(* Logix 5000 project; controller DUNEW2PLC1 vendor 1 type 14 code 221 rev 33.11; software revision 33.00 *)

TASK DUNEWINDER2 (continuous, watchdog 500 ms) : MainProgram, UnServo_9, EOT_Trip_11, Error_State_10, Latch_UnLatch_State_6_7_8, MoveXY_State_2_3, MoveZ_State_4_5, Ready_State_1, Initialize, PID_Tension_Servo
TASK SafetyTask (periodic, rate 20 ms, priority 10, watchdog 20 ms) : Safety

MODULES
   Local : vendor 1 type 14 code 221 (5069 0, rev 33.11)
      DUNEW2AMP : 2198-P031 (Ethernet 192.168.140.15, rev 11.3, A_MotionDiagnostics RPI 1 ms, B_MotionSync RPI 2 ms)
      DUNEW2SERVO2 : vendor 1 type 45 code 31 (Ethernet 192.168.140.17, rev 11.2, C_Safety_Output RPI 20 ms, B_MotionSync RPI 2 ms, D_Safety_Input RPI 10 ms, A_MotionDiagnostics RPI 1 ms)
      DUNEW2SERVO1 : vendor 1 type 45 code 31 (Ethernet 192.168.140.16, rev 11.3, C_Safety_Output RPI 20 ms, A_MotionDiagnostics RPI 1 ms, D_Safety_Input RPI 10 ms, B_MotionSync RPI 2 ms)
      DUNEW2NETSW : vendor 1 type 12 code 241 (Ethernet 192.168.140.10, rev 10.1, Output RPI 1000 ms)
      DUNE2CAM1 : vendor 678 type 100 code 274 (Ethernet 192.168.140.19, rev 11.1, Output RPI 60 ms)
       : vendor 1 type 115 code 313 (5069 5, rev 2.1, StandardDataDriven RPI 13.1 ms)
           Local:5:O.Ch00.Data   // Tension_Servo_CMD
       : 5069-IB16 (5069 2, rev 2.14, StandardDataDriven RPI 5 ms)
           Local:2:I.Pt07.Data   // O/T SWITCH OVERTRAVEL SWITCH
           Local:2:I.Pt06.Data   // TENSION ON/OFF
           Local:2:I.Pt13.Data   // Cabinet lighted push button
       : 5069-IB16 (5069 6, rev 2.14, StandardDataDriven RPI 5 ms)
       : 5069-OB16 (5069 3, rev 2.14, StandardDataDriven RPI 5 ms)
           Local:3:O.Pt01.Data   // Latching signal output
           Local:3:O.Pt11.Data   // Reset PB - Light
           Local:3:O.Pt15.Data   // Beacon - Sounder
           Local:3:O.Pt13.Data   // Beacon - Amber
           Local:3:O.Pt12.Data   // Beacon - Green
           Local:3:O.Pt14.Data   // Beacon - Red
       : 5069-OB16 (5069 7, rev 2.14, StandardDataDriven RPI 5 ms)
       : 5069-IF8 (5069 4, rev 2.11, StandardDataDriven RPI 12.5 ms)
           Local:4:I   // Wire tension (N)
       : 5069-IB16 (5069 1, rev 2.14, StandardDataDriven RPI 5 ms)
           Local:1:I.Pt08.Data   // Latch top
           Local:1:I.Pt15.Data   // The wire break switch was causing electrical problems, so we use the load-cell as a proxy for wire break
           Local:1:I.Pt09.Data   // Latch middle
      DUNEW2PLC2 : 1734-AENT (Ethernet 192.168.140.14, rev 6.12)
          : vendor 1 type 35 code 16 (PointIO 2, rev 2.1, Output RPI 20 ms, Input RPI 10 ms)
          : vendor 1 type 35 code 15 (PointIO 1, rev 2.1, Output RPI 20 ms, Input RPI 10 ms)
              DUNEW2PLC2:1:I.Pt03Data   // EStop Pullcord 1
              DUNEW2PLC2:1:I.Pt04Data   // EStop Pullcord 2
              DUNEW2PLC2:1:I.Pt02Data   // EStop Rack
              DUNEW2PLC2:1:I.Pt01Data   // LC OSS2
              DUNEW2PLC2:1:I.Pt05Data   // Run Key
              DUNEW2PLC2:1:I.Pt00Data   // LC OSS1
END_MODULES

ADD_ON_INSTRUCTION SCP   (* revision 1.0, vendor CVKI *)
// Scale with Parameters
// Help:
// Rockwell Software RSLogix 500 Description:
// The Input value is scaled to a range determined by creating a linear relationship between input min and max values and scaled min and max values. The scaled result is returned to the address indicated by the output parameter.
VAR_INPUT
   Input : REAL; {required}   // Value to be Scaled
   Input_Min : REAL; {required}   // Minimum Value for the Input
   Input_Max : REAL; {required}   // Maximum Value for the Input
   Scaled_Min : REAL; {required}   // Minimum Scaling Value
   Scaled_Max : REAL; {required}   // Maximum Scaling Value
END_VAR
VAR_OUTPUT
   Output : REAL; {access Read Only, required}   // Scaled Value [Slope*Input + Offset]
END_VAR
VAR
   offset : REAL;   // Offset Value [Scaled Min - (Input Min * Slope)]
   slope : REAL;   // Slope Value [(Scaled Max - Scaled Min)/(Input Max - Input Min)]
END_VAR

ROUTINE Logic   (* ladder *)
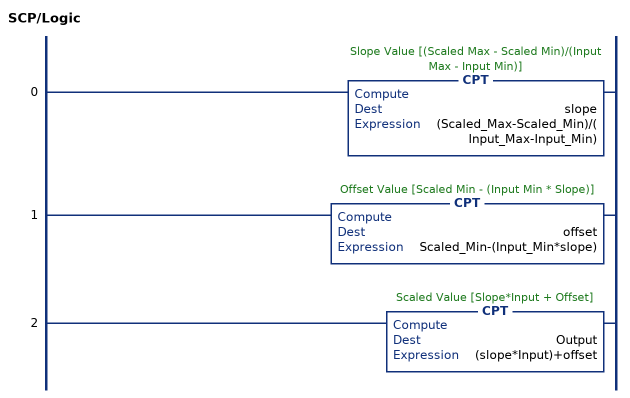
   0: CPT(slope,(Scaled_Max-Scaled_Min)/(Input_Max-Input_Min));
   1: CPT(offset,Scaled_Min-(Input_Min*slope));
   2: CPT(Output,(slope*Input)+offset);
END_ROUTINE
END_ADD_ON_INSTRUCTION

VAR_GLOBAL   (* controller tags *)
   a_actual : REAL := 700.0062;
   a_signed : REAL := -243.85713;
   accel_xy : REAL;   // Tangential acceleration of the winding head in xy-plane
   ACTUATOR_POS : DINT := 1; {access Read Only}
   AFI : BOOL;
   ALL_EOT_GOOD : BOOL := 1; {access Read Only}
   always_regulate_speed : BOOL := 1;
   APA_IS_VERTICAL : BOOL; {access Read Only}
   blink_off : TIMER := (PRE := 500, ACC := 490, EN := 1, TT := 1);
   blink_on : TIMER := (PRE := 500, ACC := 500, EN := 1, DN := 1);
   bypass_xy_move : BOOL := 1;
   CAM_F_EN : BOOL := 1;
   CAM_F_TRIGGER : BOOL := 1;
   check_tension_stable : BOOL := 1;   // Check if the tension is stable at the setpoint before moving the winding head
   current_command : REAL;
   current_command_high : REAL := 1.5; {constant}
   current_command_low : REAL := -0.5; {constant}
   DUNEW1AMP : AXIS_CIP_DRIVE;
   DUNEW2AXIS : MOTION_GROUP;
   EN_POS_TRIGGERS : BOOL;
   Enable_SFX : BOOL;
   Enable_SLS : BOOL;
   ERROR_CODE : DINT; {access Read Only}
   ESTOP : ALIAS FOR DUNEW2PLC2:1:I.Pt02Data;
   FIFO_Data : REAL[6]; {access Read Only}
   FIFO_FLUSH : BOOL;   // Flush the camera FIFOs.
   FRAME_LOC_FT_BTM : BOOL := 1;
   FRAME_LOC_FT_MID : BOOL := 1;
   FRAME_LOC_FT_TOP : BOOL := 1;
   FRAME_LOC_HD_BTM : BOOL := 1;
   FRAME_LOC_HD_MID : BOOL := 1;
   FRAME_LOC_HD_TOP : BOOL := 1;
   gamma : REAL := 20.0;
   HEAD_POS : DINT;
   HomeTrigger : BOOL;
   INIT_DONE : BOOL := 1; {access Read Only}
   INPUTS2 : ALIAS FOR Local:2:I;
   J : REAL := 2000.0;
   LATCH_ACTUATOR_BOTTOM : BOOL;
   LATCH_ACTUATOR_HOMED : BOOL; {access Read Only}
   LATCH_ACTUATOR_MID : BOOL;
   LATCH_ACTUATOR_TOP : BOOL;
   latch_ouput : ALIAS FOR Local:3:O.Pt01.Data;
   MACHINE_SW_STAT : BOOL[32] := ([1] := 1, [2] := 1, [3] := 1, [4] := 1, [6] := 1, [8] := 1, [9] := 1, [17] := 1, [18] := 1, [19] := 1, [20] := 1, [21] := 1, [25] := 1, [26] := 1, [27] := 1, [28] := 1, [29] := 1, [30] := 1, [31] := 1); {access Read Only}
   MAS : BOOL := 1;   // Motion Axis Stop
   MASTER_Z_GO : BOOL := 1; {access Read Only}
   max_tolerable_tension : REAL := 9.0;
   MAX_TOLERABLE_Z : REAL := 5.0; {constant}
   MCCD_X_Y_Axis : MOTION_INSTRUCTION := (FLAGS := 33554432);
   MCCD_X_Y_Axis1 : MOTION_INSTRUCTION := (FLAGS := 33554432);
   MINUS_X_EOT : BOOL := 1; {access Read Only}
   MINUS_Y_EOT : BOOL := 1; {access Read Only}
   MORE_STATS : BOOL[32]; {access Read Only}
   MORE_STATS_S : BOOL[32] := ([0] := 1);
   MOVE_TYPE : INT;   // 0 = No Move 1 = XY JOG 2 = XY Plane Move 3 = Z JOG 4 = Z Axis Move 5 = Toggle Latch Actuator 6 = Home the Latch Actuator 7 = Unlock Latch Actuator Motor 8 = Un-Servo Motors 9 = PLC_Init
   neutral_cv : REAL := 2.5;
   NEXTSTATE : DINT := 1; {access Read Only}
   overtension_timer : TIMER := (PRE := 100);
   pid_cv_high_limit : REAL := 10.0;
   pid_cv_low_limit : REAL;
   pid_cv_out : REAL := 2.5;
   PID_LOOP_TIMER : TIMER := (PRE := 5, ACC := 4, EN := 1, TT := 1);
   pid_loop_timer_bypass : BOOL;
   pid_start_bias : BOOL;
   PLUS_X_EOT : BOOL := 1; {access Read Only}
   PLUS_Y_EOT : BOOL := 1; {access Read Only}
   POSITION : REAL[1,2]; {constant}
   READ_FIFOS : BOOL;
   ResetPB : BOOL;
   resetPB_S : BOOL;
   ROT_LOC_KEY : AB:1769_DI32:I:0; {access Read Only}
   Run_Alarm : BOOL;
   Safety_Reset_FallingEdge : BOOL;
   Safety_System_Healthy : BOOL := 1;
   Safety_Tripped_S : BOOL;
   SetPoint_CV : REAL;
   SetPoint_Override : REAL;
   SetPoint_PV : REAL := 2.3567553;   // wire tension from load cell (N)
   SLS_Active_Limit : REAL := 50.0;
   SLS_Request1 : BOOL;
   speed_regulator_switch : BOOL := 1;   // This is our "enable safe speed" switch, repurposed to switch the speed regulator
   STATE : DINT := 1; {access Read Only}   // CURRENT State Machine State
   STATE6_IND : BOOL; {access Read Only}
   STATE8_IND : BOOL := 1; {access Read Only}
   T01 : TIMER := (PRE := 5000, ACC := 5000, EN := 1, DN := 1);
   tension : ALIAS FOR Local:4:I.Ch01.Data;   // wire tension (N)
   TENSION_CONTROL_OK : BOOL;
   tension_limited_speed : REAL;
   tension_motor_out : ALIAS FOR Local:5:O.Ch00.Data;
   TENSION_ON_SWITCH : BOOL;
   tension_on_switch_delay_on_start : TIMER := (PRE := 1000);
   tension_setpoint : REAL := 6.25;
   tension_stabilizing : BOOL := 1;
   tension_stable_timer : TIMER := (PRE := 200);
   v_0 : REAL := 0.049999997;
   v_xy : REAL;   // velocity of winding head in xy plane
   v_xyz : REAL;   // Velocity of winding head in xyz space
   winding_head_pid : PID := (CTL := 41984, INI := 1, OLL := 1, DVNA := 1, SP := 2.0, KP := 0.1, KI := 0.4, KD := 0.1, MAXS := 10.0, MAXO := 100.0, UPD := 0.05, PV := 2.3567543, ERR := -0.3567543, PVH := 10.0, MAXI := 10.0, MAXCV := 10.0, MAXTIE := 10.0, DATA[0] := 0.20484047, DATA[1] := -377.08075, DATA[2] := 2.3567543, DATA[3] := -0.3567543, DATA[4] := 2.0, DATA[5] := 10.0, DATA[6] := 1.0, DATA[7] := 0.90000004, DATA[8] := 0.1, DATA[9] := 0.4, DATA[10] := 0.1, DATA[11] := 0.1, DATA[12] := 0.4, DATA[13] := 0.1, DATA[15] := 0.1, DATA[16] := 10.0);
   wire_break_proxy : BOOL;
   wire_break_tension : REAL := 2.5;
   X_axis : AXIS_CIP_DRIVE; {access Read Only}
   X_Axis_SFX : SAFETY_FEEDBACK_INTERFACE := (FeedbackValid := 1, O1 := 1, PositionScaling := 512.0, FeedbackResolution := 512, Unwind := 512, FaultType := 1, PositionScalingOut := 512.0, UnwindOut := 512);
   X_Axis_SLS : SAFELY_LIMITED_SPEED := (RestartType := 1, ColdStartType := 1, O1 := 1, CheckDelay := 3000, ActiveLimit := 10.0, FaultType := 1);
   X_DELTA : REAL;
   X_PARKED : BOOL; {access Read Only}
   X_POSITION : ALIAS FOR POSITION[0,0]; {constant}
   X_SPEED : REAL;
   X_XFER_OK : BOOL; {access Read Only}   // If at the head, check head support arms. Same for foot
   X_Y : COORDINATE_SYSTEM;
   XY_ACCELERATION : REAL := 150.0;   // Maximum positive acceleration for position move.
   XY_DECEL_REQ : REAL;
   XY_DECELERATION : REAL := 300.0;   // Maximum negative acceleration for position move.
   XY_MAX_ACCELERATION : REAL;   // Maximum positive acceleration for position move.
   XY_MAX_DECELERATION : REAL;   // Maximum negative acceleration for position move.
   XY_MAX_VELOCITY : REAL;   // Maximum velocity for position move.
   xy_regulated_acceleration : REAL := 2000.0;
   xy_regulated_deceleration : REAL := 2000.0;
   XY_SPEED : REAL := 300.0;   // Maximum velocity for position move.
   XY_SPEED_REQ : REAL := 300.0;   // XY Requested speed copy of XY_Speed to be used for MCLM and MCCD in MoveXY
   Y_axis : AXIS_CIP_DRIVE; {access Read Only}
   Y_DELTA : REAL := 5.75;
   Y_MOUNT_XFER_OK : BOOL; {access Read Only}
   Y_POSITION : ALIAS FOR POSITION[0,1]; {constant}
   Y_SPEED : REAL;
   Y_XFER_OK : BOOL := 1; {access Read Only}
   Y_Xfer_Window_Btm : BOOL;
   Y_Xfer_Window_Mid : BOOL;
   Y_Xfer_Window_Top : BOOL;
   Z_ACCELERATION : REAL := 600.0;
   Z_axis : AXIS_CIP_DRIVE; {access Read Only}
   Z_DECELLERATION : REAL := 600.0;
   Z_EOT : BOOL := 1; {access Read Only}
   Z_EXTENDED : BOOL; {access Read Only}
   Z_FIXED_LATCHED : BOOL; {access Read Only}
   Z_FIXED_PRESENT : BOOL; {access Read Only}
   Z_OK_TO_ENGAGE : BOOL; {access Read Only}
   Z_POSITION : REAL;
   Z_RETRACTED : BOOL := 1; {access Read Only}
   Z_SAFE_TO_WITHDRAW : BOOL;
   Z_SPEED : REAL;
   Z_STAGE_LATCHED : BOOL := 1; {access Read Only}
   Z_STAGE_PRESENT : BOOL := 1; {access Read Only}   // Winding head is on the Z-arm
   Z_STAGE_UNLATCHED : BOOL; {access Read Only}
END_VAR

PROGRAM Camera   (* main routine CameraControl *)
// Controls to capture data from the Cognex camera.
VAR
   Cam_F_InspectionRes_0 : REAL[32]; {access Read Only}
   Cam_F_InspectionRes_1 : REAL[10]; {access Read Only}
   Cam_F_InspectionRes_2 : REAL[10]; {access Read Only}
   Cam_F_InspectionRes_3 : REAL[10]; {access Read Only}
   FIFO_CTRL : CONTROL[6] := ([0].LEN := 10, [0].EM := 1, [1].LEN := 10, [1].EM := 1, [2].LEN := 10, [2].EM := 1, [3].LEN := 10, [3].EM := 1, [4].LEN := 10, [4].EM := 1, [5].LEN := 10, [5].EM := 1); {access Read Only}
   foundIt : BOOL; {access Read Only}
   LightRing : TIMER := (PRE := 100); {access Read Only}
   Manual_Trig : BOOL; {access Read Only}
   osob : BOOL[32]; {access Read Only}
   ossb : BOOL[32] := ([3] := 1); {access Read Only}
   Pos_trigger : BOOL := 1; {access Read Only}
   RegistrationData : MOTION_INSTRUCTION[8] := ([0].FLAGS := -1845493760, [0].EN := 1, [0].ER := 1, [0].ERR := 3, [1].FLAGS := -1845493760, [1].EN := 1, [1].ER := 1, [1].ERR := 3); {access Read Only}
   triggerOneShotOB : BOOL; {access Read Only}
   triggerOneShotSB : BOOL := 1; {access Read Only}
   TriggerResetTimer1 : TIMER := (PRE := 100, ACC := 5, EN := 1, TT := 1); {access Read Only}
   TriggerResetTimer2 : TIMER := (PRE := 100); {access Read Only}
   X_axis_Cam_F_Pos : REAL[10]; {access Read Only}
   X_axis_Cam_F_Position : REAL := -5.1799655; {access Read Only}
   x_pos : REAL := 564.005; {access Read Only}
   x_pos_next : REAL := 564.005;
   Y_axis_Cam_F_Pos : REAL[10]; {access Read Only}
   Y_axis_Cam_F_Position : REAL := 12.123628; {access Read Only}
   y_pos : REAL := 2465.8398;
   y_pos_next : REAL := 2465.8398;
END_VAR

ROUTINE CameraControl   (* ladder *)
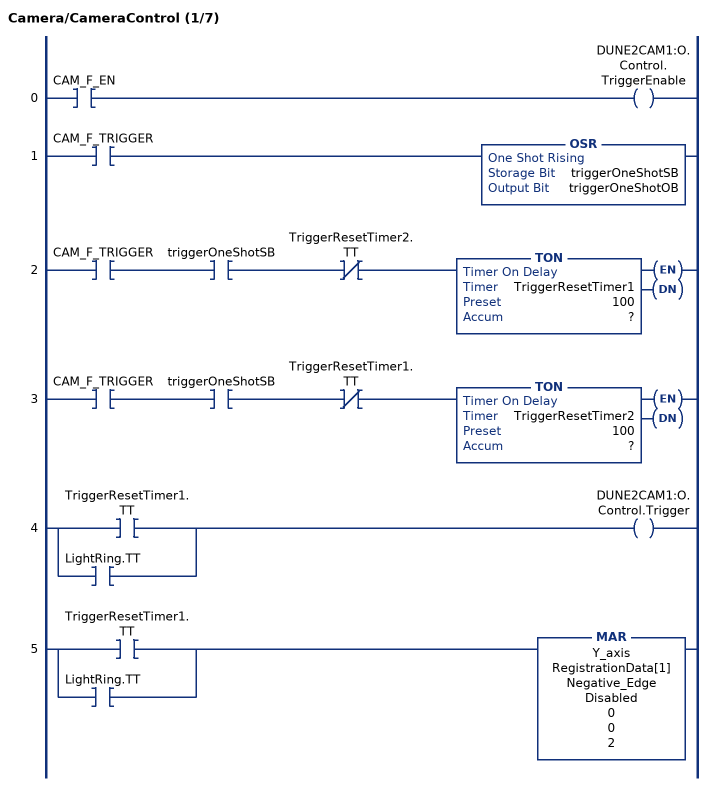
   0: XIC(CAM_F_EN)OTE(DUNE2CAM1:O.Control.TriggerEnable);
   1: XIC(CAM_F_TRIGGER)OSR(triggerOneShotSB,triggerOneShotOB);
   2: XIC(CAM_F_TRIGGER)XIC(triggerOneShotSB)XIO(TriggerResetTimer2.TT)TON(TriggerResetTimer1,?,?);
   3: XIC(CAM_F_TRIGGER)XIC(triggerOneShotSB)XIO(TriggerResetTimer1.TT)TON(TriggerResetTimer2,?,?);
   4: [XIC(TriggerResetTimer1.TT) ,XIC(LightRing.TT) ]OTE(DUNE2CAM1:O.Control.Trigger);
   5: [XIC(TriggerResetTimer1.TT) ,XIC(LightRing.TT) ]MAR(Y_axis,RegistrationData[1],Negative_Edge,Disabled,0,0,2);
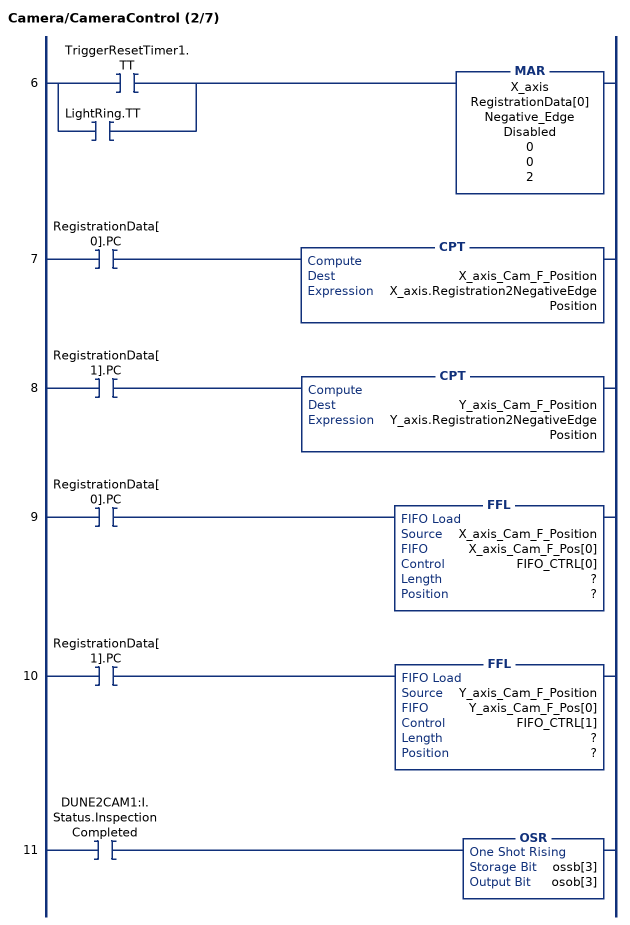
   6: [XIC(TriggerResetTimer1.TT) ,XIC(LightRing.TT) ]MAR(X_axis,RegistrationData[0],Negative_Edge,Disabled,0,0,2);
   7: XIC(RegistrationData[0].PC)CPT(X_axis_Cam_F_Position,X_axis.Registration2NegativeEdgePosition);
   8: XIC(RegistrationData[1].PC)CPT(Y_axis_Cam_F_Position,Y_axis.Registration2NegativeEdgePosition);
   9: XIC(RegistrationData[0].PC)FFL(X_axis_Cam_F_Position,X_axis_Cam_F_Pos[0],FIFO_CTRL[0],?,?);
   10: XIC(RegistrationData[1].PC)FFL(Y_axis_Cam_F_Position,Y_axis_Cam_F_Pos[0],FIFO_CTRL[1],?,?);
   11: XIC(DUNE2CAM1:I.Status.InspectionCompleted)OSR(ossb[3],osob[3]);
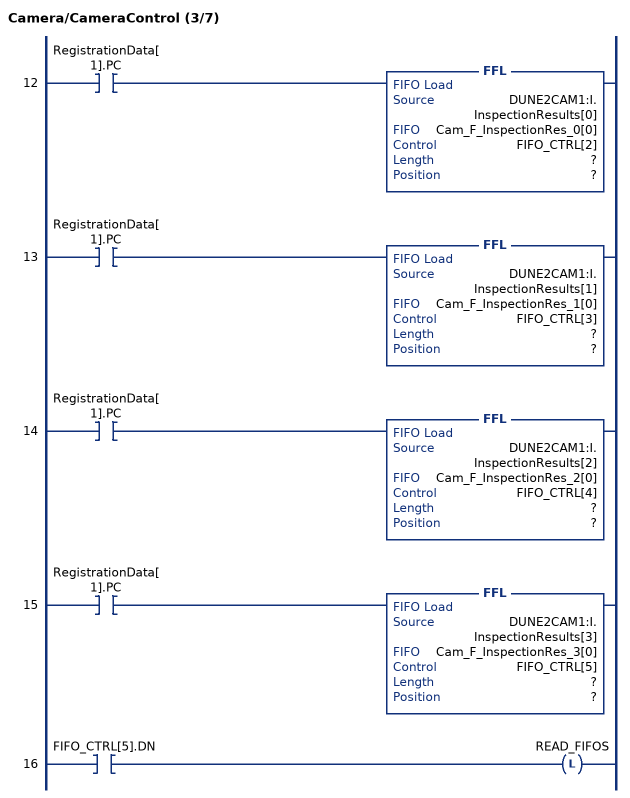
   12: XIC(RegistrationData[1].PC)FFL(DUNE2CAM1:I.InspectionResults[0],Cam_F_InspectionRes_0[0],FIFO_CTRL[2],?,?);
   13: XIC(RegistrationData[1].PC)FFL(DUNE2CAM1:I.InspectionResults[1],Cam_F_InspectionRes_1[0],FIFO_CTRL[3],?,?);
   14: XIC(RegistrationData[1].PC)FFL(DUNE2CAM1:I.InspectionResults[2],Cam_F_InspectionRes_2[0],FIFO_CTRL[4],?,?);
   15: XIC(RegistrationData[1].PC)FFL(DUNE2CAM1:I.InspectionResults[3],Cam_F_InspectionRes_3[0],FIFO_CTRL[5],?,?);
   16: XIC(FIFO_CTRL[5].DN)OTL(READ_FIFOS);
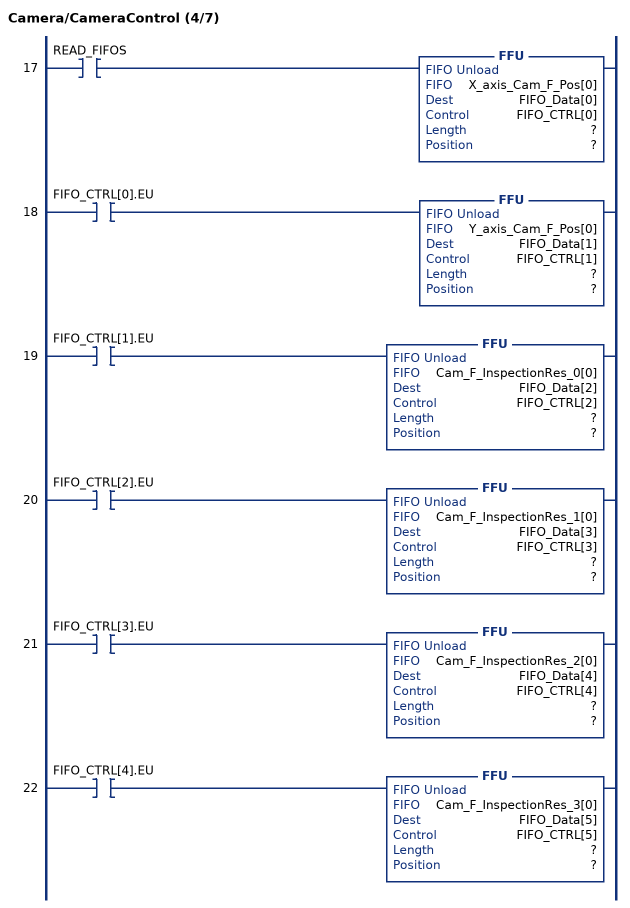
   17: XIC(READ_FIFOS)FFU(X_axis_Cam_F_Pos[0],FIFO_Data[0],FIFO_CTRL[0],?,?);
   18: XIC(FIFO_CTRL[0].EU)FFU(Y_axis_Cam_F_Pos[0],FIFO_Data[1],FIFO_CTRL[1],?,?);
   19: XIC(FIFO_CTRL[1].EU)FFU(Cam_F_InspectionRes_0[0],FIFO_Data[2],FIFO_CTRL[2],?,?);
   20: XIC(FIFO_CTRL[2].EU)FFU(Cam_F_InspectionRes_1[0],FIFO_Data[3],FIFO_CTRL[3],?,?);
   21: XIC(FIFO_CTRL[3].EU)FFU(Cam_F_InspectionRes_2[0],FIFO_Data[4],FIFO_CTRL[4],?,?);
   22: XIC(FIFO_CTRL[4].EU)FFU(Cam_F_InspectionRes_3[0],FIFO_Data[5],FIFO_CTRL[5],?,?);
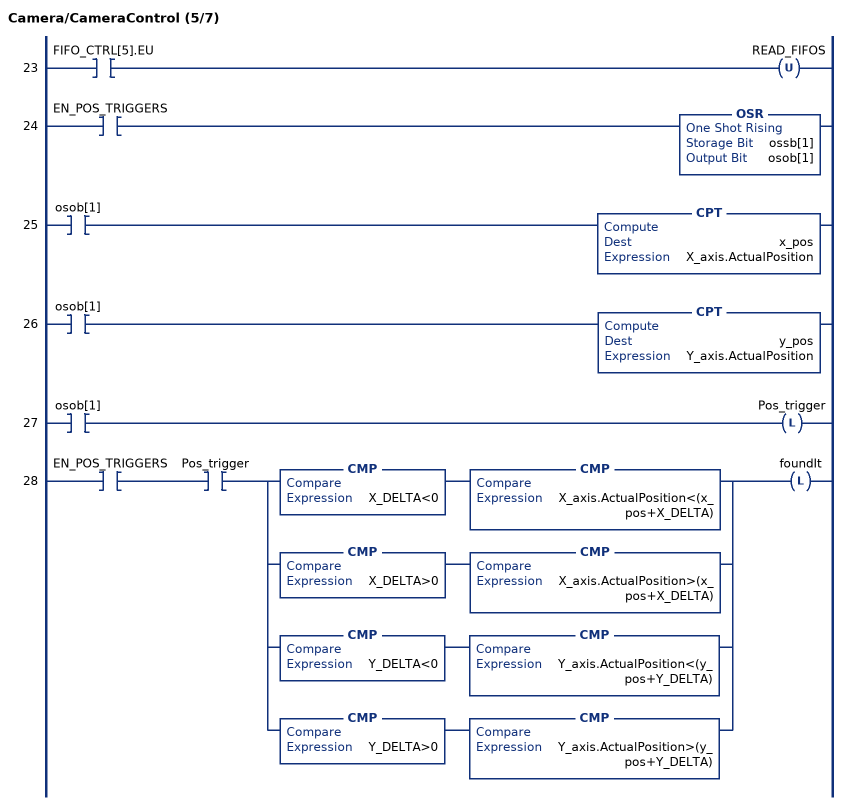
   23: XIC(FIFO_CTRL[5].EU)OTU(READ_FIFOS);
   24: XIC(EN_POS_TRIGGERS)OSR(ossb[1],osob[1]);
   25: XIC(osob[1])CPT(x_pos,X_axis.ActualPosition);
   26: XIC(osob[1])CPT(y_pos,Y_axis.ActualPosition);
   27: XIC(osob[1])OTL(Pos_trigger);
   28: XIC(EN_POS_TRIGGERS)XIC(Pos_trigger)[[CMP(X_DELTA<0) CMP(X_axis.ActualPosition<(x_pos+X_DELTA)) ,CMP(X_DELTA>0) CMP(X_axis.ActualPosition>(x_pos+X_DELTA)) ] ,[CMP(Y_DELTA<0) CMP(Y_axis.ActualPosition<(y_pos+Y_DELTA)) ,CMP(Y_DELTA>0) CMP(Y_axis.ActualPosition>(y_pos+Y_DELTA)) ] ]OTL(foundIt);
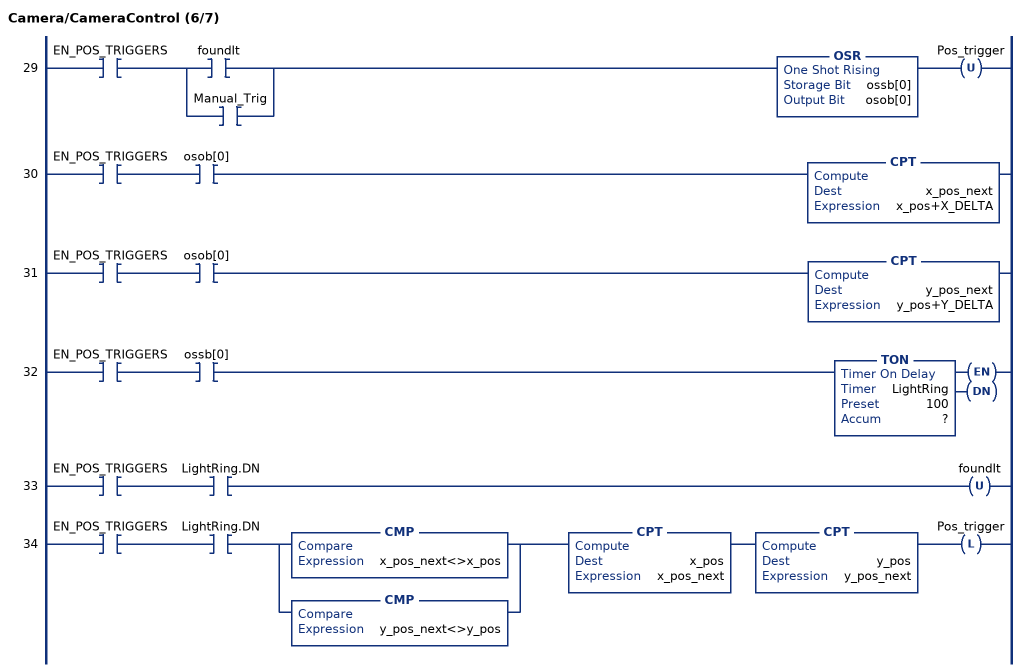
   29: XIC(EN_POS_TRIGGERS)[XIC(foundIt) ,XIC(Manual_Trig) ]OSR(ossb[0],osob[0])OTU(Pos_trigger);
   30: XIC(EN_POS_TRIGGERS)XIC(osob[0])CPT(x_pos_next,x_pos+X_DELTA);
   31: XIC(EN_POS_TRIGGERS)XIC(osob[0])CPT(y_pos_next,y_pos+Y_DELTA);
   32: XIC(EN_POS_TRIGGERS)XIC(ossb[0])TON(LightRing,?,?);
   33: XIC(EN_POS_TRIGGERS)XIC(LightRing.DN)OTU(foundIt);
   34: XIC(EN_POS_TRIGGERS)XIC(LightRing.DN)[CMP(x_pos_next<>x_pos) ,CMP(y_pos_next<>y_pos) ]CPT(x_pos,x_pos_next)CPT(y_pos,y_pos_next)OTL(Pos_trigger);
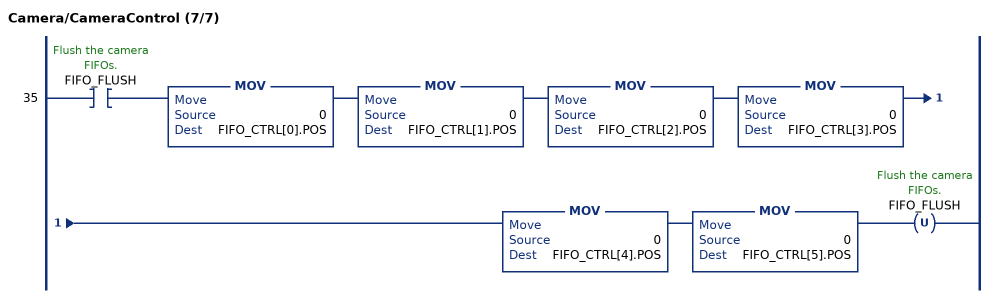
   35: XIC(FIFO_FLUSH)MOV(0,FIFO_CTRL[0].POS)MOV(0,FIFO_CTRL[1].POS)MOV(0,FIFO_CTRL[2].POS)MOV(0,FIFO_CTRL[3].POS)MOV(0,FIFO_CTRL[4].POS)MOV(0,FIFO_CTRL[5].POS)OTU(FIFO_FLUSH);
END_ROUTINE
END_PROGRAM

PROGRAM EOT_Trip_11   (* main routine EOT_TRIP *)
VAR
   AXIS_STAT : MOTION_INSTRUCTION[32] := ([0].FLAGS := 33554432, [1].FLAGS := 33554432, [2].FLAGS := 33554432, [3].FLAGS := 33554432, [4].FLAGS := 33554432, [5].FLAGS := 570425344, [5].DN := 1, [6].FLAGS := 570425344, [6].DN := 1, [7].FLAGS := 570425344, [7].DN := 1, [7].STATUS := 2, [7].STATE := 3, [8].FLAGS := 33554432, [9].FLAGS := 570425344, [9].DN := 1, [9].STATUS := 2, [9].STATE := 3, [10].FLAGS := -1845493760, [10].EN := 1, [10].ER := 1, [10].ERR := 5, [11].FLAGS := 268435456, [11].ER := 1, [11].ERR := 3, [11].STATUS := 2, [12].FLAGS := 33554432, [13].FLAGS := 704643072, [13].DN := 1, [13].PC := 1, [20].FLAGS := 704643072, [20].DN := 1, [20].PC := 1, [29].FLAGS := 33554432, [30].FLAGS := 33554432, [31].FLAGS := 33554432); {access Read Only}
   oneshotob : BOOL[32]; {access Read Only}
   oneshotsb : BOOL[32] := ([12] := 1, [13] := 1, [14] := 1, [15] := 1); {access Read Only}
   STATE11_IND : BOOL; {access Read Only}
END_VAR

ROUTINE EOT_TRIP   (* ladder *)
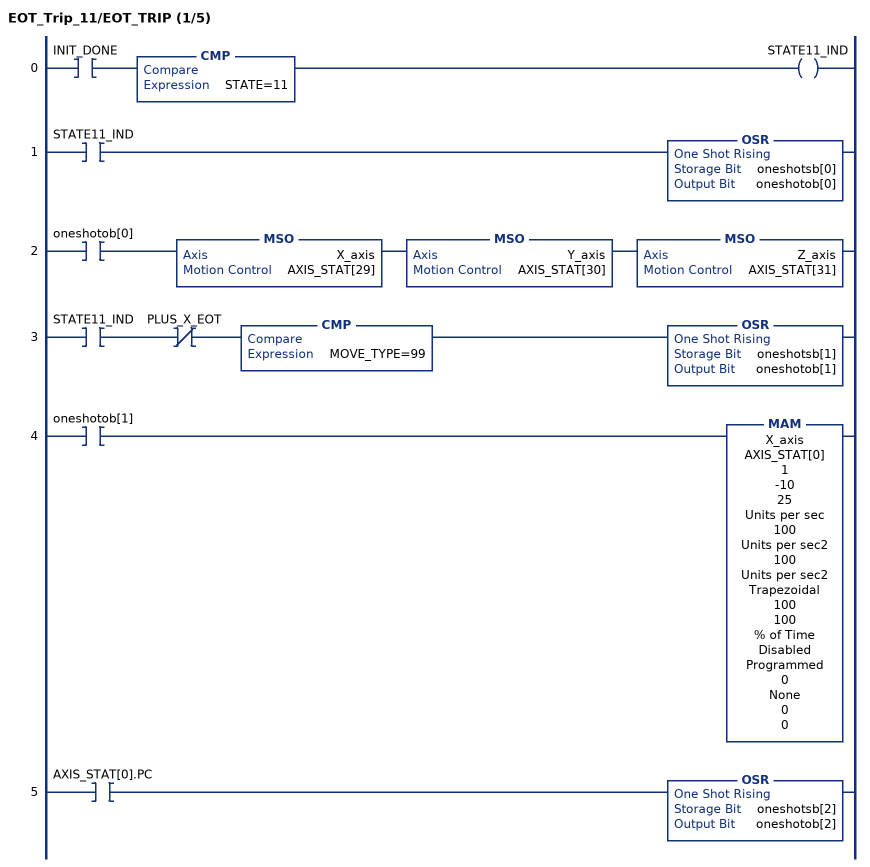
   0: XIC(INIT_DONE)CMP(STATE=11)OTE(STATE11_IND);
   1: XIC(STATE11_IND)OSR(oneshotsb[0],oneshotob[0]);
   2: XIC(oneshotob[0])MSO(X_axis,AXIS_STAT[29])MSO(Y_axis,AXIS_STAT[30])MSO(Z_axis,AXIS_STAT[31]);
   3: XIC(STATE11_IND)XIO(PLUS_X_EOT)CMP(MOVE_TYPE=99)OSR(oneshotsb[1],oneshotob[1]);
   4: XIC(oneshotob[1])MAM(X_axis,AXIS_STAT[0],1,-10,25,Units per sec,100,Units per sec2,100,Units per sec2,Trapezoidal,100,100,% of Time,Disabled,Programmed,0,None,0,0);
   5: XIC(AXIS_STAT[0].PC)OSR(oneshotsb[2],oneshotob[2]);
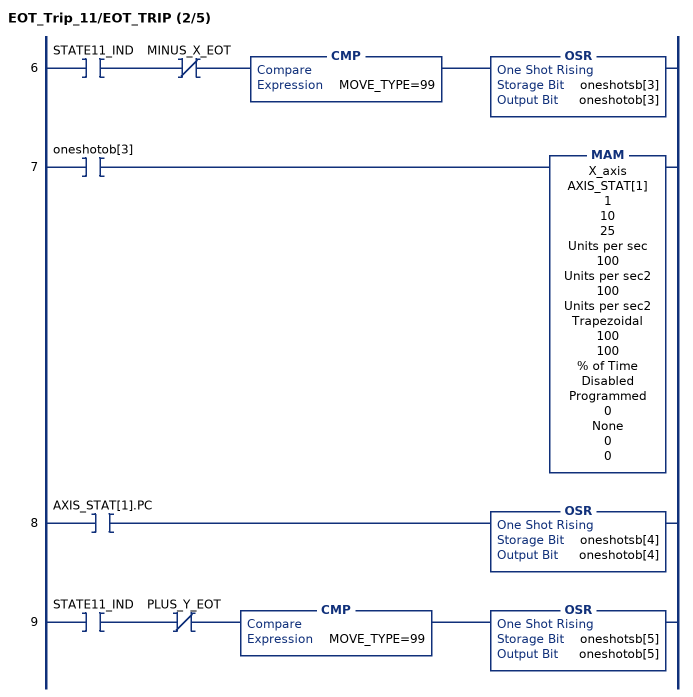
   6: XIC(STATE11_IND)XIO(MINUS_X_EOT)CMP(MOVE_TYPE=99)OSR(oneshotsb[3],oneshotob[3]);
   7: XIC(oneshotob[3])MAM(X_axis,AXIS_STAT[1],1,10,25,Units per sec,100,Units per sec2,100,Units per sec2,Trapezoidal,100,100,% of Time,Disabled,Programmed,0,None,0,0);
   8: XIC(AXIS_STAT[1].PC)OSR(oneshotsb[4],oneshotob[4]);
   9: XIC(STATE11_IND)XIO(PLUS_Y_EOT)CMP(MOVE_TYPE=99)OSR(oneshotsb[5],oneshotob[5]);
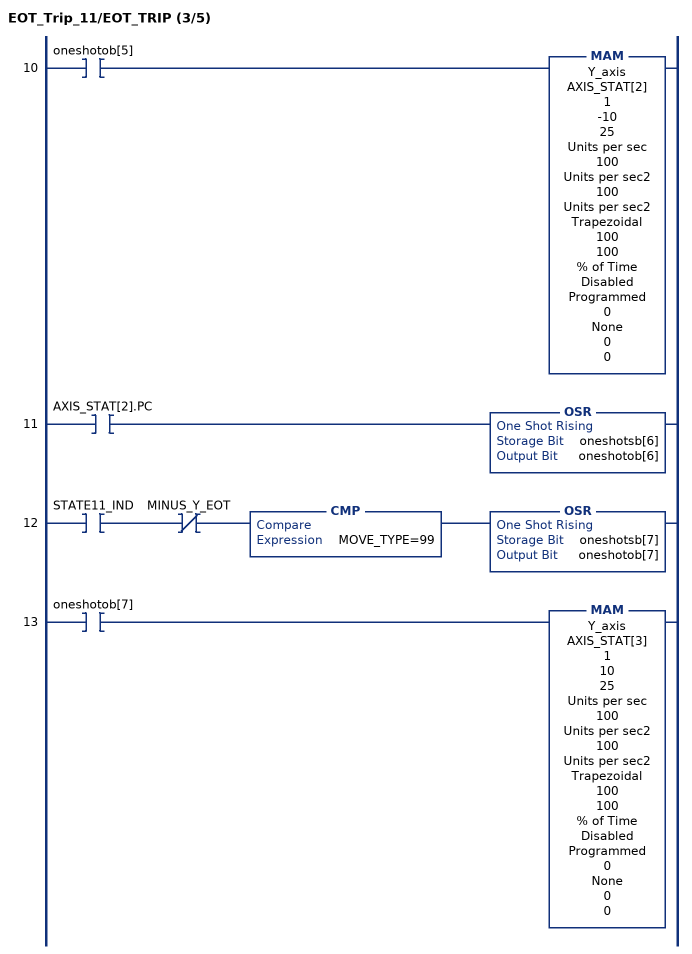
   10: XIC(oneshotob[5])MAM(Y_axis,AXIS_STAT[2],1,-10,25,Units per sec,100,Units per sec2,100,Units per sec2,Trapezoidal,100,100,% of Time,Disabled,Programmed,0,None,0,0);
   11: XIC(AXIS_STAT[2].PC)OSR(oneshotsb[6],oneshotob[6]);
   12: XIC(STATE11_IND)XIO(MINUS_Y_EOT)CMP(MOVE_TYPE=99)OSR(oneshotsb[7],oneshotob[7]);
   13: XIC(oneshotob[7])MAM(Y_axis,AXIS_STAT[3],1,10,25,Units per sec,100,Units per sec2,100,Units per sec2,Trapezoidal,100,100,% of Time,Disabled,Programmed,0,None,0,0);
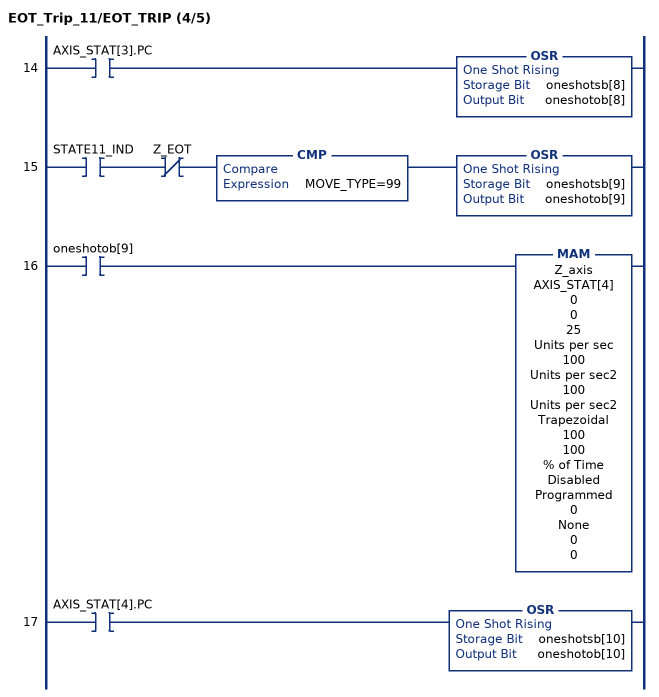
   14: XIC(AXIS_STAT[3].PC)OSR(oneshotsb[8],oneshotob[8]);
   15: XIC(STATE11_IND)XIO(Z_EOT)CMP(MOVE_TYPE=99)OSR(oneshotsb[9],oneshotob[9]);
   16: XIC(oneshotob[9])MAM(Z_axis,AXIS_STAT[4],0,0,25,Units per sec,100,Units per sec2,100,Units per sec2,Trapezoidal,100,100,% of Time,Disabled,Programmed,0,None,0,0);
   17: XIC(AXIS_STAT[4].PC)OSR(oneshotsb[10],oneshotob[10]);
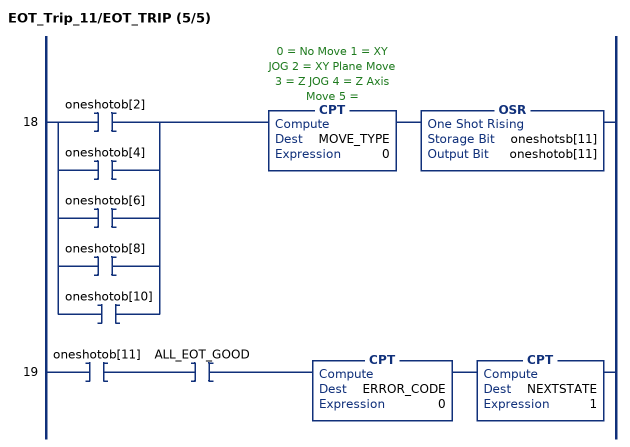
   18: [XIC(oneshotob[2]) ,XIC(oneshotob[4]) ,XIC(oneshotob[6]) ,XIC(oneshotob[8]) ,XIC(oneshotob[10]) ]CPT(MOVE_TYPE,0)OSR(oneshotsb[11],oneshotob[11]);
   19: XIC(oneshotob[11])XIC(ALL_EOT_GOOD)CPT(ERROR_CODE,0)CPT(NEXTSTATE,1);
END_ROUTINE
END_PROGRAM

PROGRAM Error_State_10   (* main routine Error *)
VAR
   oneshotob : BOOL[32]; {access Read Only}
        [0]   // On entry to state 6 or 7
   oneshotsb : BOOL[32]; {access Read Only}
        [0]   // While in state 6 or 7
   STATE10_IND : BOOL; {access Read Only}
   TIMEOUT : BOOL; {access Read Only}
   X_AXIS_STAT : MOTION_INSTRUCTION[32] := ([0].FLAGS := 33554432, [3].FLAGS := 33554432, [4].FLAGS := 33554432); {access Read Only}
   Y_AXIS_STAT : MOTION_INSTRUCTION[32] := ([0].FLAGS := 704643072, [0].DN := 1, [0].PC := 1, [3].FLAGS := 33554432, [4].FLAGS := 33554432); {access Read Only}
   Z_AXIS_STAT : MOTION_INSTRUCTION[32] := ([0].FLAGS := 33554432, [3].FLAGS := 33554432, [4].FLAGS := 33554432, [5].FLAGS := 33554432, [6].FLAGS := 33554432); {access Read Only}
END_VAR

ROUTINE Error   (* ladder *)
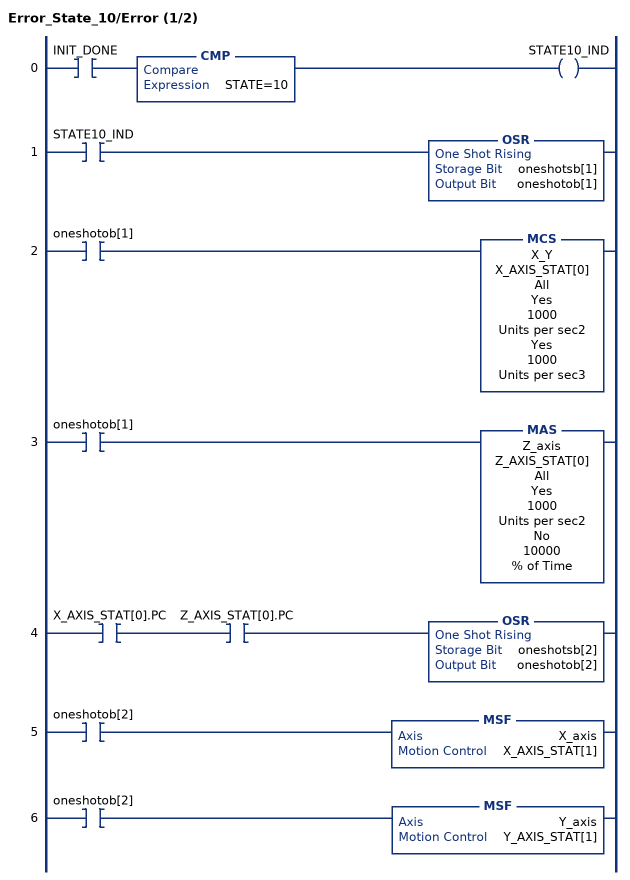
   0: XIC(INIT_DONE)CMP(STATE=10)OTE(STATE10_IND);
   1: XIC(STATE10_IND)OSR(oneshotsb[1],oneshotob[1]);
   2: XIC(oneshotob[1])MCS(X_Y,X_AXIS_STAT[0],All,Yes,1000,Units per sec2,Yes,1000,Units per sec3);
   3: XIC(oneshotob[1])MAS(Z_axis,Z_AXIS_STAT[0],All,Yes,1000,Units per sec2,No,10000,% of Time);
   4: XIC(X_AXIS_STAT[0].PC)XIC(Z_AXIS_STAT[0].PC)OSR(oneshotsb[2],oneshotob[2]);
   5: XIC(oneshotob[2])MSF(X_axis,X_AXIS_STAT[1]);
   6: XIC(oneshotob[2])MSF(Y_axis,Y_AXIS_STAT[1]);
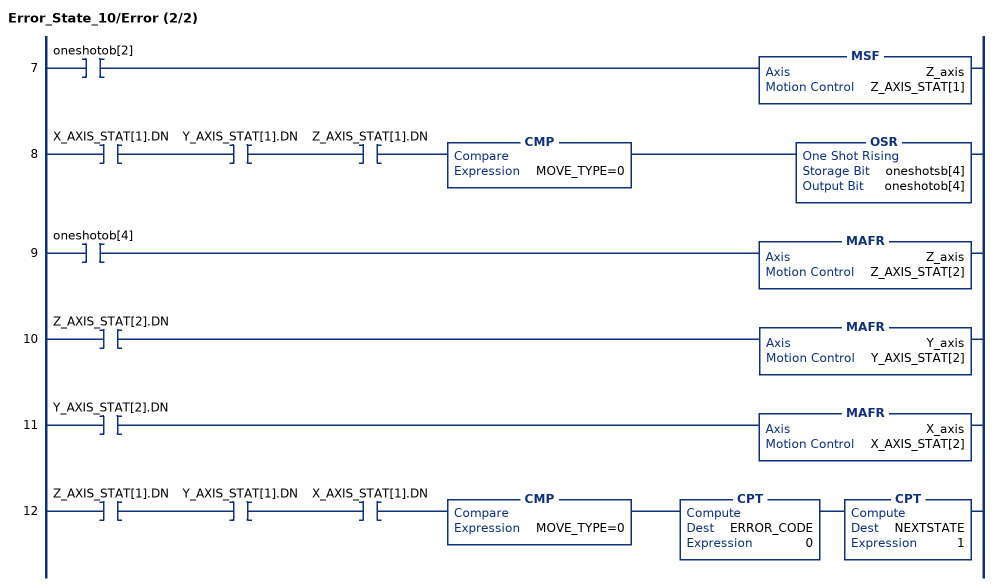
   7: XIC(oneshotob[2])MSF(Z_axis,Z_AXIS_STAT[1]);
   8: XIC(X_AXIS_STAT[1].DN)XIC(Y_AXIS_STAT[1].DN)XIC(Z_AXIS_STAT[1].DN)CMP(MOVE_TYPE=0)OSR(oneshotsb[4],oneshotob[4]);
   9: XIC(oneshotob[4])MAFR(Z_axis,Z_AXIS_STAT[2]);
   10: XIC(Z_AXIS_STAT[2].DN)MAFR(Y_axis,Y_AXIS_STAT[2]);
   11: XIC(Y_AXIS_STAT[2].DN)MAFR(X_axis,X_AXIS_STAT[2]);
   12: XIC(Z_AXIS_STAT[1].DN)XIC(Y_AXIS_STAT[1].DN)XIC(X_AXIS_STAT[1].DN)CMP(MOVE_TYPE=0)CPT(ERROR_CODE,0)CPT(NEXTSTATE,1);
END_ROUTINE
END_PROGRAM

PROGRAM Initialize   (* main routine Init *)
// First state to set up machine
VAR
   INIT_SW : BOOL := 1;
   OutBit : BOOL[32]; {access Read Only}
   SetBit : BOOL[32] := ([0] := 1); {access Read Only}
   TIMER : TIMER := (PRE := 2000, ACC := 2000, EN := 1, DN := 1);
   Z_AXIS_STAT : MOTION_INSTRUCTION[32] := ([0].FLAGS := 301989888, [0].ER := 1, [0].ERR := 11); {access Read Only}
END_VAR

ROUTINE Init   (* ladder *)
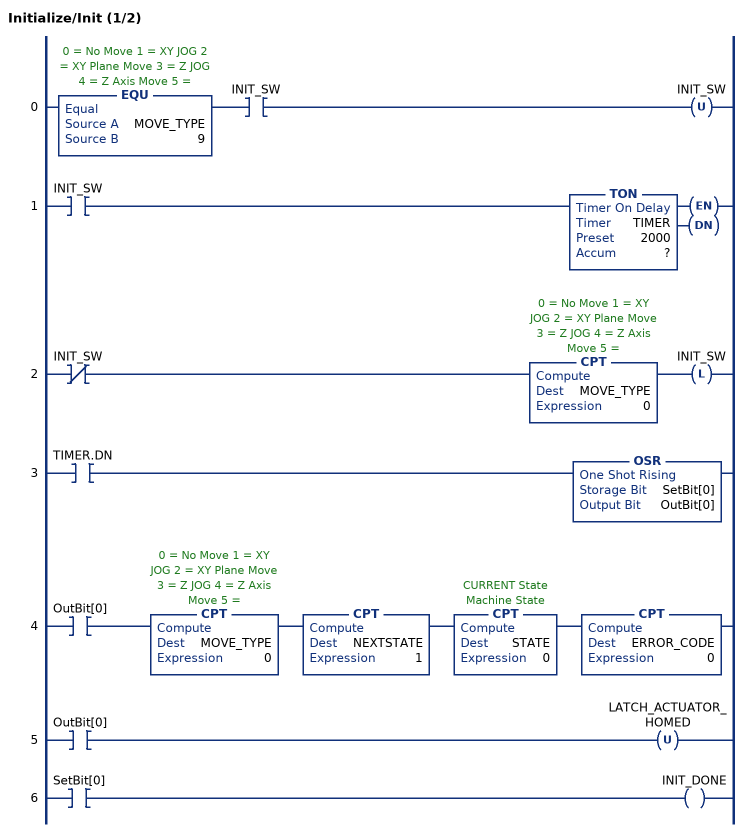
   0: EQU(MOVE_TYPE,9)XIC(INIT_SW)OTU(INIT_SW);
   1: XIC(INIT_SW)TON(TIMER,?,?);
   2: XIO(INIT_SW)CPT(MOVE_TYPE,0)OTL(INIT_SW);
   3: XIC(TIMER.DN)OSR(SetBit[0],OutBit[0]);
   4: XIC(OutBit[0])CPT(MOVE_TYPE,0)CPT(NEXTSTATE,1)CPT(STATE,0)CPT(ERROR_CODE,0);
   5: XIC(OutBit[0])OTU(LATCH_ACTUATOR_HOMED);
   6: XIC(SetBit[0])OTE(INIT_DONE);
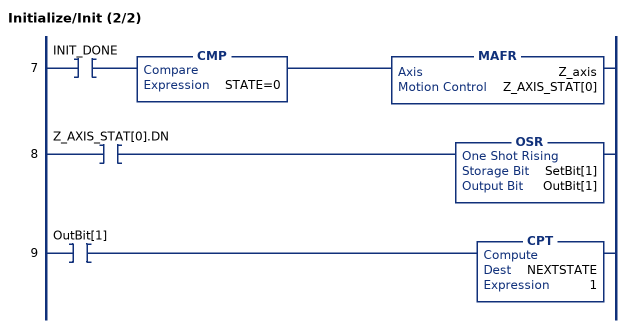
   7: XIC(INIT_DONE)CMP(STATE=0)MAFR(Z_axis,Z_AXIS_STAT[0]);
   8: XIC(Z_AXIS_STAT[0].DN)OSR(SetBit[1],OutBit[1]);
   9: XIC(OutBit[1])CPT(NEXTSTATE,1);
END_ROUTINE
END_PROGRAM

PROGRAM Latch_UnLatch_State_6_7_8   (* main routine Latch_Driver *)
VAR
   Delay_Fixed_Latched : TIMER := (PRE := 100);
   Delay_Z_Latched : TIMER := (PRE := 100, ACC := 100, EN := 1, DN := 1);
   ENABLE_ACTUATOR : BOOL; {access Read Only}
   HomeCounter : COUNTER := (PRE := 20, ACC := 20, DN := 1); {access Read Only}
   HomeSignal : BOOL; {access Read Only}
   HomeTimer1 : TIMER := (PRE := 300); {access Read Only}
   HomeTimer2 : TIMER := (PRE := 300); {access Read Only}
   LatchCounter2 : COUNTER := (PRE := 2, ACC := 2, DN := 1); {access Read Only}
   LatchCounter3 : COUNTER := (PRE := 2, ACC := 2, DN := 1); {access Read Only}
   Latching_pulse_duration : TIMER := (PRE := 50); {access Read Only}
   Latching_pulse_interval : TIMER := (PRE := 200);
   LatchingTimeoutCounter : COUNTER := (PRE := 10, ACC := 1);   // When you enter state 6 or 7, start counting seconds
   LatchTimer3 : TIMER := (PRE := 250); {access Read Only}
   LatchTimer4 : TIMER := (PRE := 250); {access Read Only}
   LatchTimer5 : TIMER := (PRE := 250); {access Read Only}
   LatchTimer6 : TIMER := (PRE := 250); {access Read Only}
   oneshotob : BOOL[32]; {access Read Only}
        [1]   // For one scan, when we enter state 6 and actuator is enabled
        [9]   // Entered state 6 but the actuator was not enabled
   oneshotsb : BOOL[32] := ([5] := 1, [7] := 1, [10] := 1); {access Read Only}
        [1]   // While in state 6 and operator is enabled
        [8]   // While in state 6
        [6]   // LatchCounter done
        [2]   // Latch successfully moved to the next position
   PREV_ACT_POS : DINT := 2; {access Read Only}   // Store the previous actuator position
   STATE7_IND : BOOL; {access Read Only}
   TimeoutTimer1 : TIMER := (PRE := 1000);
   TimeoutTimer2 : TIMER := (PRE := 1000);
   UNLOCK_LATCH_MOTOR_SHAFT : BOOL := 1; {access Read Only}
END_VAR

ROUTINE Latch_Driver   (* ladder *)
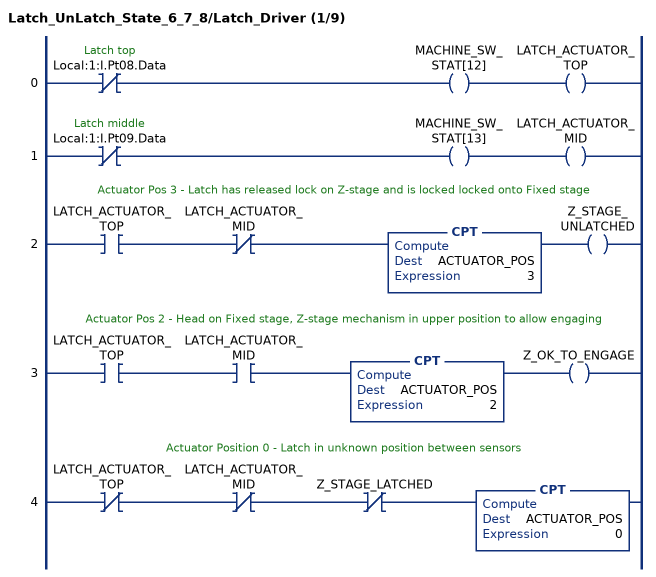
   0: XIO(Local:1:I.Pt08.Data)OTE(MACHINE_SW_STAT[12])OTE(LATCH_ACTUATOR_TOP);
   1: XIO(Local:1:I.Pt09.Data)OTE(MACHINE_SW_STAT[13])OTE(LATCH_ACTUATOR_MID);
   // Actuator Pos 3 - Latch has released lock on Z-stage and is locked locked onto Fixed stage
   2: XIC(LATCH_ACTUATOR_TOP)XIO(LATCH_ACTUATOR_MID)CPT(ACTUATOR_POS,3)OTE(Z_STAGE_UNLATCHED);
   // Actuator Pos 2 - Head on Fixed stage, Z-stage mechanism in upper position to allow engaging
   3: XIC(LATCH_ACTUATOR_TOP)XIC(LATCH_ACTUATOR_MID)CPT(ACTUATOR_POS,2)OTE(Z_OK_TO_ENGAGE);
   // Actuator Position 0 - Latch in unknown position between sensors
   4: XIO(LATCH_ACTUATOR_TOP)XIO(LATCH_ACTUATOR_MID)XIO(Z_STAGE_LATCHED)CPT(ACTUATOR_POS,0);
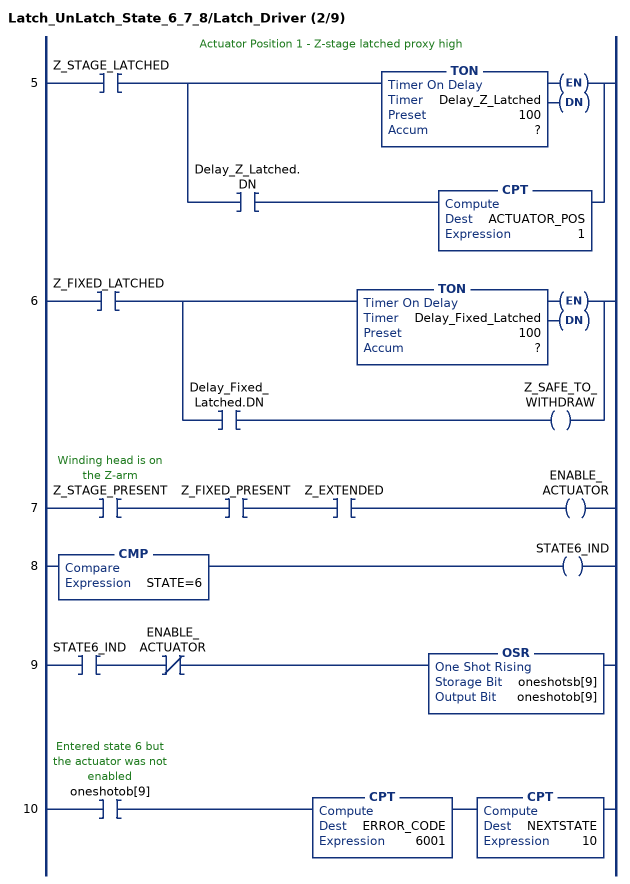
   // Actuator Position 1 - Z-stage latched proxy high
   5: XIC(Z_STAGE_LATCHED)[TON(Delay_Z_Latched,?,?) ,XIC(Delay_Z_Latched.DN) CPT(ACTUATOR_POS,1) ];
   6: XIC(Z_FIXED_LATCHED)[TON(Delay_Fixed_Latched,?,?) ,XIC(Delay_Fixed_Latched.DN) OTE(Z_SAFE_TO_WITHDRAW) ];
   7: XIC(Z_STAGE_PRESENT)XIC(Z_FIXED_PRESENT)XIC(Z_EXTENDED)OTE(ENABLE_ACTUATOR);
   8: CMP(STATE=6)OTE(STATE6_IND);
   9: XIC(STATE6_IND)XIO(ENABLE_ACTUATOR)OSR(oneshotsb[9],oneshotob[9]);
   10: XIC(oneshotob[9])CPT(ERROR_CODE,6001)CPT(NEXTSTATE,10);
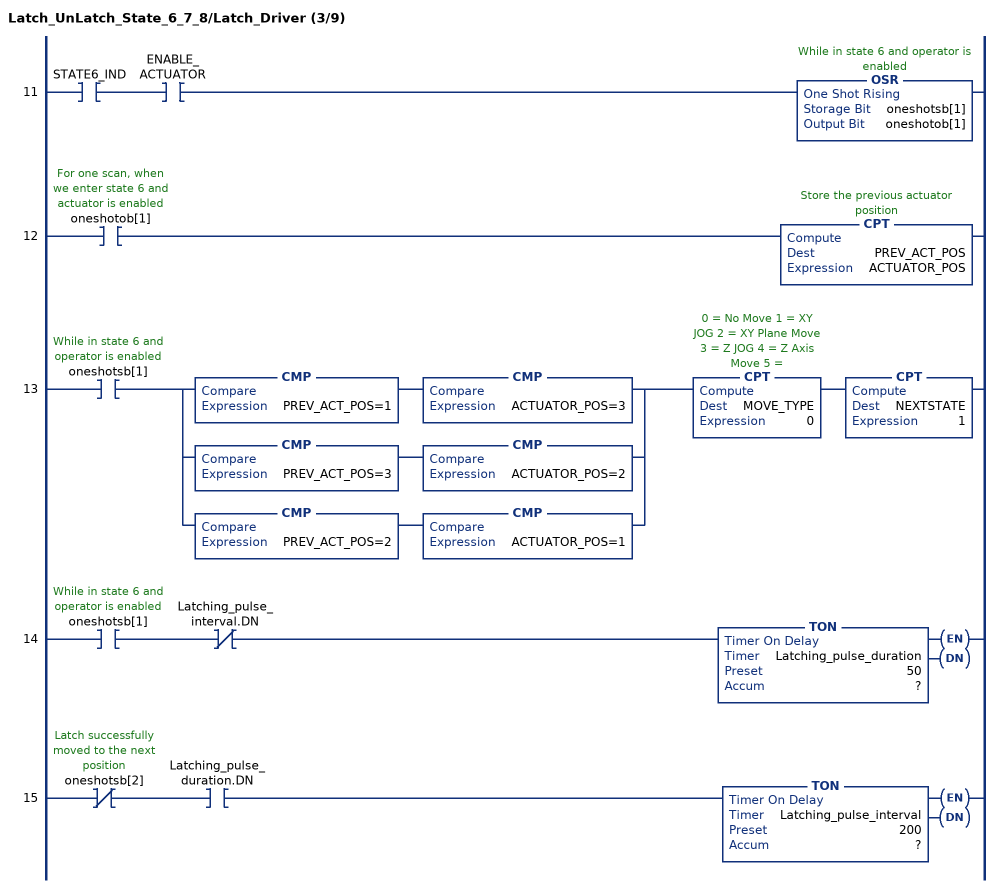
   11: XIC(STATE6_IND)XIC(ENABLE_ACTUATOR)OSR(oneshotsb[1],oneshotob[1]);
   12: XIC(oneshotob[1])CPT(PREV_ACT_POS,ACTUATOR_POS);
   13: XIC(oneshotsb[1])[CMP(PREV_ACT_POS=1) CMP(ACTUATOR_POS=3) ,CMP(PREV_ACT_POS=3) CMP(ACTUATOR_POS=2) ,CMP(PREV_ACT_POS=2) CMP(ACTUATOR_POS=1) ]CPT(MOVE_TYPE,0)CPT(NEXTSTATE,1);
   14: XIC(oneshotsb[1])XIO(Latching_pulse_interval.DN)TON(Latching_pulse_duration,?,?);
   15: XIO(oneshotsb[2])XIC(Latching_pulse_duration.DN)TON(Latching_pulse_interval,?,?);
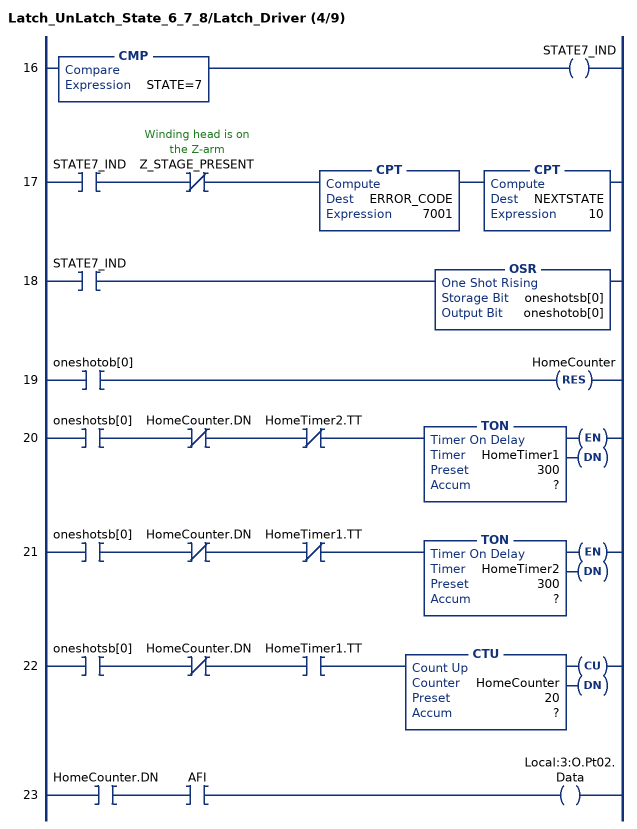
   16: CMP(STATE=7)OTE(STATE7_IND);
   17: XIC(STATE7_IND)XIO(Z_STAGE_PRESENT)CPT(ERROR_CODE,7001)CPT(NEXTSTATE,10);
   18: XIC(STATE7_IND)OSR(oneshotsb[0],oneshotob[0]);
   19: XIC(oneshotob[0])RES(HomeCounter);
   20: XIC(oneshotsb[0])XIO(HomeCounter.DN)XIO(HomeTimer2.TT)TON(HomeTimer1,?,?);
   21: XIC(oneshotsb[0])XIO(HomeCounter.DN)XIO(HomeTimer1.TT)TON(HomeTimer2,?,?);
   22: XIC(oneshotsb[0])XIO(HomeCounter.DN)XIC(HomeTimer1.TT)CTU(HomeCounter,?,?);
   23: XIC(HomeCounter.DN)XIC(AFI)OTE(Local:3:O.Pt02.Data);
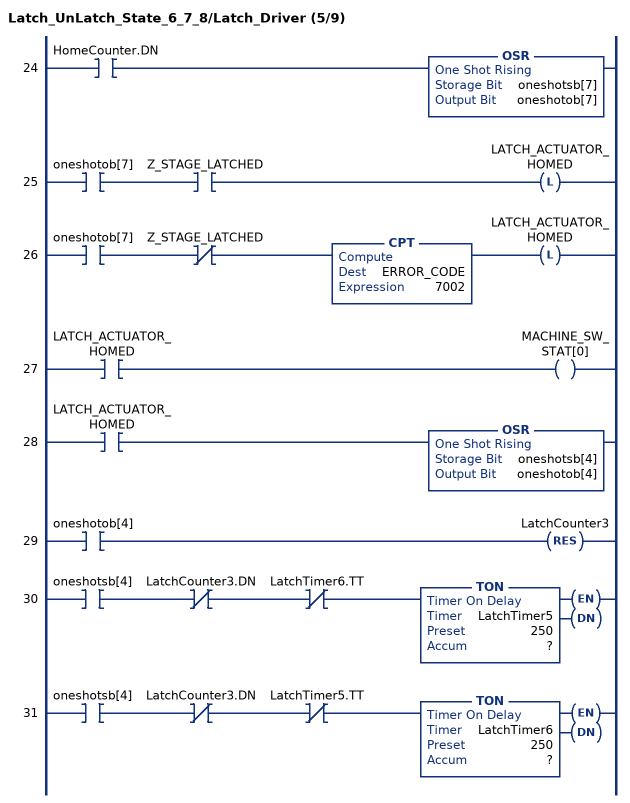
   24: XIC(HomeCounter.DN)OSR(oneshotsb[7],oneshotob[7]);
   25: XIC(oneshotob[7])XIC(Z_STAGE_LATCHED)OTL(LATCH_ACTUATOR_HOMED);
   26: XIC(oneshotob[7])XIO(Z_STAGE_LATCHED)CPT(ERROR_CODE,7002)OTL(LATCH_ACTUATOR_HOMED);
   27: XIC(LATCH_ACTUATOR_HOMED)OTE(MACHINE_SW_STAT[0]);
   28: XIC(LATCH_ACTUATOR_HOMED)OSR(oneshotsb[4],oneshotob[4]);
   29: XIC(oneshotob[4])RES(LatchCounter3);
   30: XIC(oneshotsb[4])XIO(LatchCounter3.DN)XIO(LatchTimer6.TT)TON(LatchTimer5,?,?);
   31: XIC(oneshotsb[4])XIO(LatchCounter3.DN)XIO(LatchTimer5.TT)TON(LatchTimer6,?,?);
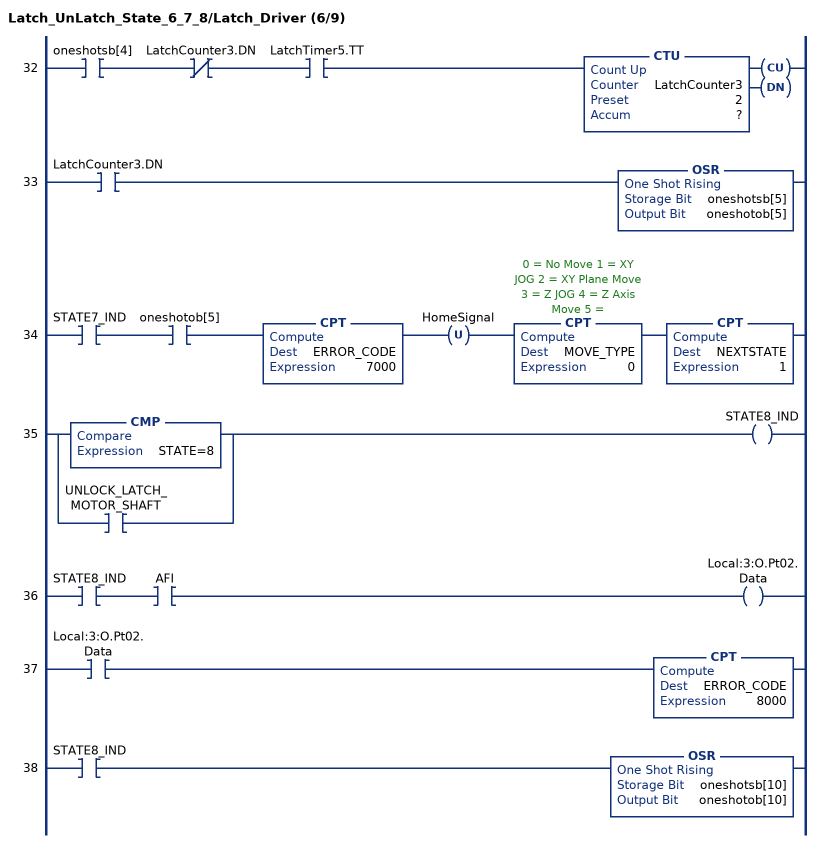
   32: XIC(oneshotsb[4])XIO(LatchCounter3.DN)XIC(LatchTimer5.TT)CTU(LatchCounter3,?,?);
   33: XIC(LatchCounter3.DN)OSR(oneshotsb[5],oneshotob[5]);
   34: XIC(STATE7_IND)XIC(oneshotob[5])CPT(ERROR_CODE,7000)OTU(HomeSignal)CPT(MOVE_TYPE,0)CPT(NEXTSTATE,1);
   35: [CMP(STATE=8) ,XIC(UNLOCK_LATCH_MOTOR_SHAFT) ]OTE(STATE8_IND);
   36: XIC(STATE8_IND)XIC(AFI)OTE(Local:3:O.Pt02.Data);
   37: XIC(Local:3:O.Pt02.Data)CPT(ERROR_CODE,8000);
   38: XIC(STATE8_IND)OSR(oneshotsb[10],oneshotob[10]);
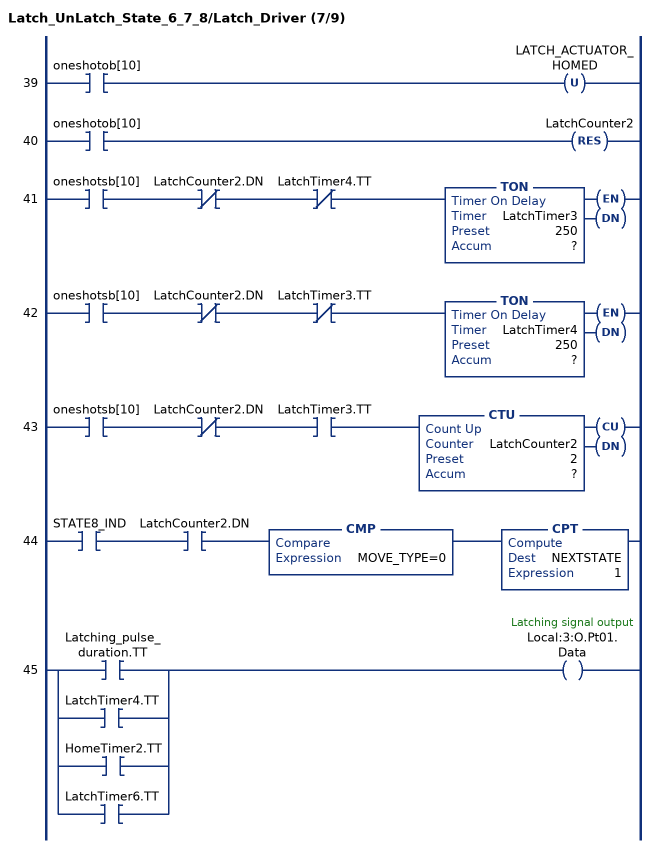
   39: XIC(oneshotob[10])OTU(LATCH_ACTUATOR_HOMED);
   40: XIC(oneshotob[10])RES(LatchCounter2);
   41: XIC(oneshotsb[10])XIO(LatchCounter2.DN)XIO(LatchTimer4.TT)TON(LatchTimer3,?,?);
   42: XIC(oneshotsb[10])XIO(LatchCounter2.DN)XIO(LatchTimer3.TT)TON(LatchTimer4,?,?);
   43: XIC(oneshotsb[10])XIO(LatchCounter2.DN)XIC(LatchTimer3.TT)CTU(LatchCounter2,?,?);
   44: XIC(STATE8_IND)XIC(LatchCounter2.DN)CMP(MOVE_TYPE=0)CPT(NEXTSTATE,1);
   45: [XIC(Latching_pulse_duration.TT) ,XIC(LatchTimer4.TT) ,XIC(HomeTimer2.TT) ,XIC(LatchTimer6.TT) ]OTE(Local:3:O.Pt01.Data);
